FUNCTION_BLOCK FB_ModBusExample

VAR
	fbReadCoil : FB_MBReadCoils;
	nReadValue : BYTE;
END_VAR

fbReadCoil(
	sIPAddr:= '172.22.1.14', 
	nTCPPort:= 502 , 
	nUnitID:=16#FF , 
	nQuantity:= 1, 
	nMBAddr:= 0, 
	cbLength:= SIZEOF(nReadValue), 
	pDestAddr:= ADR(nReadValue) , 
	bExecute:= TRUE, 
	tTimeout:= , 
	bBusy=> , 
	bError=> , 
	nErrId=> , 
	cbRead=> );

END_FUNCTION_BLOCK

(* stored: Version 1.1.0.1, ProductVersion 3.1.4024.16
   POU FB_ModBusExample: Id {ce5a885b-c4f4-47d9-b1de-e3517741924d}, SpecialFunc None *)
